// TIA Portal V17 export
// export: Created 2022-07-20T06:59:38.9365482Z, ExportSetting WithDefaults, DisplayName Totally Integrated Automation Portal, DisplayVersion V17, DisplayName TIA Portal Openness, DisplayVersion V17, DisplayName TIA Portal Version Control Interface, DisplayVersion V17, DisplayName SINAMICS Startdrive Advanced, DisplayVersion V17, DisplayName SINAMICS Startdrive G130, G150, S120, S150, SINAMICS MV, S210, DisplayVersion V17, DisplayName SINAMICS Startdrive G110M, G120, G120C, G120D, G120P, G115D, DisplayVersion V17, DisplayName STEP 7 Professional, DisplayVersion V17, DisplayName STEP 7 Safety, DisplayVersion V17, DisplayName WinCC Advanced, DisplayVersion V17
FUNCTION_BLOCK "FB10011_WordToBoolAT"   // FB10011, LAD
TITLE = FB10011_WordToBoolAT
{ S7_Optimized_Access := 'TRUE' }
AUTHOR : Jonathan
FAMILY : 1001x_CONVERT
VERSION : 1.0
// Release note : 
// 1.0 - Feature developped
// stored: AutoNumber false, IsIECCheckEnabled false, IsRetainMemResEnabled false, MemoryReserve 100, SetENOAutomatically false, UDAEnableTagReadback false
   VAR_INPUT
      conveyor { ExternalAccessible := 'False'; ExternalVisible := 'False'; ExternalWritable := 'False'} : Word;
   END_VAR
   VAR_OUTPUT
      motor0 { ExternalAccessible := 'False'; ExternalVisible := 'False'; ExternalWritable := 'False'} : Bool;
      motor1 { ExternalAccessible := 'False'; ExternalVisible := 'False'; ExternalWritable := 'False'} : Bool;
      motor2 { ExternalAccessible := 'False'; ExternalVisible := 'False'; ExternalWritable := 'False'} : Bool;
      motor3 { ExternalAccessible := 'False'; ExternalVisible := 'False'; ExternalWritable := 'False'} : Bool;
      motor4 { ExternalAccessible := 'False'; ExternalVisible := 'False'; ExternalWritable := 'False'} : Bool;
      motor5 { ExternalAccessible := 'False'; ExternalVisible := 'False'; ExternalWritable := 'False'} : Bool;
      motor6 { ExternalAccessible := 'False'; ExternalVisible := 'False'; ExternalWritable := 'False'} : Bool;
      motor7 { ExternalAccessible := 'False'; ExternalVisible := 'False'; ExternalWritable := 'False'} : Bool;
      motor8 { ExternalAccessible := 'False'; ExternalVisible := 'False'; ExternalWritable := 'False'} : Bool;
      motor9 { ExternalAccessible := 'False'; ExternalVisible := 'False'; ExternalWritable := 'False'} : Bool;
      motor10 { ExternalAccessible := 'False'; ExternalVisible := 'False'; ExternalWritable := 'False'} : Bool;
      motor11 { ExternalAccessible := 'False'; ExternalVisible := 'False'; ExternalWritable := 'False'} : Bool;
      motor12 { ExternalAccessible := 'False'; ExternalVisible := 'False'; ExternalWritable := 'False'} : Bool;
      motor13 { ExternalAccessible := 'False'; ExternalVisible := 'False'; ExternalWritable := 'False'} : Bool;
      motor14 { ExternalAccessible := 'False'; ExternalVisible := 'False'; ExternalWritable := 'False'} : Bool;
      motor15 { ExternalAccessible := 'False'; ExternalVisible := 'False'; ExternalWritable := 'False'} : Bool;
   END_VAR
   VAR DB_SPECIFIC
      statConveyor : Word;
   END_VAR
   VAR
      statMotors AT statConveyor : Array[0..15] of Bool;
   END_VAR
BEGIN

REGION Network 1
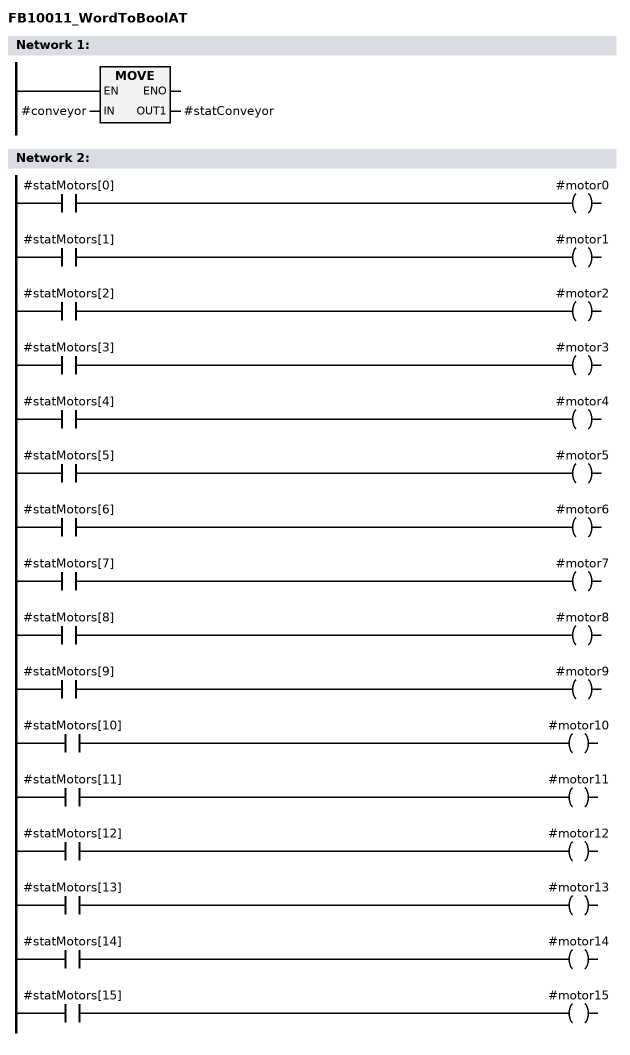
   RUNG wire#powerrail
      { S7_GenerateENO := "TRUE" } Move(in := #conveyor, out1 => #statConveyor)
   END_RUNG
   // the same network as SCL:
   #statConveyor := #conveyor;
END_REGION

REGION Network 2
   RUNG wire#powerrail
      Contact( #statMotors[0] )
      Coil( #motor0 )
   END_RUNG
   RUNG wire#powerrail
      Contact( #statMotors[1] )
      Coil( #motor1 )
   END_RUNG
   RUNG wire#powerrail
      Contact( #statMotors[2] )
      Coil( #motor2 )
   END_RUNG
   RUNG wire#powerrail
      Contact( #statMotors[3] )
      Coil( #motor3 )
   END_RUNG
   RUNG wire#powerrail
      Contact( #statMotors[4] )
      Coil( #motor4 )
   END_RUNG
   RUNG wire#powerrail
      Contact( #statMotors[5] )
      Coil( #motor5 )
   END_RUNG
   RUNG wire#powerrail
      Contact( #statMotors[6] )
      Coil( #motor6 )
   END_RUNG
   RUNG wire#powerrail
      Contact( #statMotors[7] )
      Coil( #motor7 )
   END_RUNG
   RUNG wire#powerrail
      Contact( #statMotors[8] )
      Coil( #motor8 )
   END_RUNG
   RUNG wire#powerrail
      Contact( #statMotors[9] )
      Coil( #motor9 )
   END_RUNG
   RUNG wire#powerrail
      Contact( #statMotors[10] )
      Coil( #motor10 )
   END_RUNG
   RUNG wire#powerrail
      Contact( #statMotors[11] )
      Coil( #motor11 )
   END_RUNG
   RUNG wire#powerrail
      Contact( #statMotors[12] )
      Coil( #motor12 )
   END_RUNG
   RUNG wire#powerrail
      Contact( #statMotors[13] )
      Coil( #motor13 )
   END_RUNG
   RUNG wire#powerrail
      Contact( #statMotors[14] )
      Coil( #motor14 )
   END_RUNG
   RUNG wire#powerrail
      Contact( #statMotors[15] )
      Coil( #motor15 )
   END_RUNG
   // the same network as SCL:
   #motor0 := #statMotors[0];
   #motor1 := #statMotors[1];
   #motor2 := #statMotors[2];
   #motor3 := #statMotors[3];
   #motor4 := #statMotors[4];
   #motor5 := #statMotors[5];
   #motor6 := #statMotors[6];
   #motor7 := #statMotors[7];
   #motor8 := #statMotors[8];
   #motor9 := #statMotors[9];
   #motor10 := #statMotors[10];
   #motor11 := #statMotors[11];
   #motor12 := #statMotors[12];
   #motor13 := #statMotors[13];
   #motor14 := #statMotors[14];
   #motor15 := #statMotors[15];
END_REGION
END_FUNCTION_BLOCK
